TYPE TcoCvirII_Results :
STRUCT
	{attribute addProperty Name "<#Torque#>"}
	Torque : REAL;			
	{attribute addProperty Name "<#Torque trend#>"}
	TorqueTrend : INT;			
	{attribute addProperty Name "<#Angle#>"}
	Angle : REAL;			
	{attribute addProperty Name "<#Angle trend#>"}
	AngleTrend : INT;
END_STRUCT
END_TYPE

(* stored: Version 1.1.0.1
   DUT TcoCvirII_Results: Id {49a6aa01-ce91-4905-89c4-de8a18392bec} *)
